(* CoDeSys 2.3 library: CLOCK_PLS.lib *)
(* Libraries: STANDARD.LIB 5.6.98 11:03:02 *)

(* POU MAIN, LD *)
PROGRAM MAIN
VAR
END_VAR
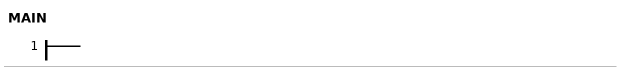
_LD_ (* Ladder Diagram *)
NETWORK 1
	*
_END_LD_
(* the same logic as Structured Text *)
(* Network 1 *)
END_PROGRAM

(* POU CLOCK_PLS, LD *)
FUNCTION_BLOCK CLOCK_PLS
VAR_INPUT
	INT_TIME_ms : INT;

END_VAR
VAR_OUTPUT
	CLOCK_PLS_BOOL: BOOL;
END_VAR
VAR
	T0: TON;
	T1: TON;
	M0: BOOL;
	M1: BOOL;
	D0: TIME;
	D1: TIME;
END_VAR
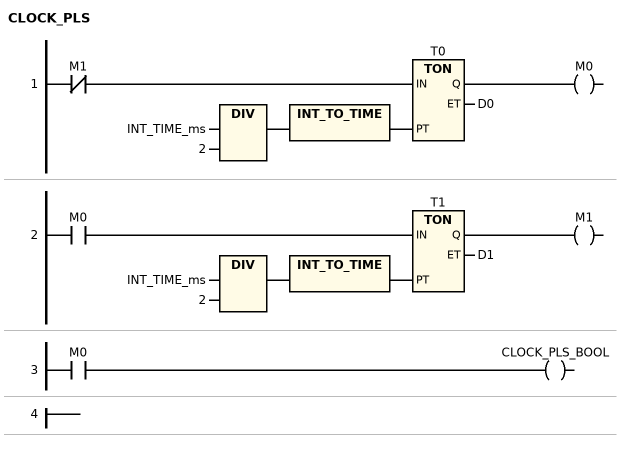
_LD_ (* Ladder Diagram *)
NETWORK 1
	[/M1] - T0:TON(IN: *, PT: INT_TO_TIME(DIV(INT_TIME_ms, 2)), ET => D0) --- (M0)
NETWORK 2
	[M0] - T1:TON(IN: *, PT: INT_TO_TIME(DIV(INT_TIME_ms, 2)), ET => D1) --- (M1)
NETWORK 3
	[M0] --- (CLOCK_PLS_BOOL)
NETWORK 4
	*
_END_LD_
(* the same logic as Structured Text *)
(* Network 1 *)
T0(IN := NOT M1, PT := INT_TO_TIME(INT_TIME_ms / 2));
D0 := T0.ET;
M0 := T0.Q;
(* Network 2 *)
T1(IN := M0, PT := INT_TO_TIME(INT_TIME_ms / 2));
D1 := T1.ET;
M1 := T1.Q;
(* Network 3 *)
CLOCK_PLS_BOOL := M0;
(* Network 4 *)
END_FUNCTION_BLOCK
